{attribute 'qualified_only'}
{attribute 'strict'}
TYPE EFeedbackMsgEd12dss :
(
	ShutterIrisPositionMsg := 10
);
END_TYPE

(* stored: Version 1.1.0.1, ProductVersion 3.1.4024.3
   DUT EFeedbackMsgEd12dss: Id {e0f35226-c5cf-40b8-91f8-632e11ab9641} *)
